FUNCTION_BLOCK AX_TON (* standard timer function block (on-delay timing) *)
  (* Standard: 61499-2; Classification: standard timer function block; Description: Copyright (c) 2024 HR Agrartechnik GmbH This program and the accompanying materials are made available under the terms of the Eclipse Public License 2.0 which is available at https://www.eclipse.org/legal/epl-2.0/ SPDX-License-Identifier: EPL-2.0 *)
  (* Version 3.0, 2025-04-14, Patrick Aigner, changed package *)
  (* Version 1.0, 2024-03-04, Franz Hoepfinger, HR Agrartechnik GmbH *)
  PACKAGE adapter::events::unidirectional::timers;
  IMPORT eclipse4diac::core::TypeHash;
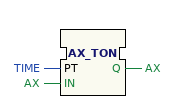
  VAR_INPUT
    PT : TIME; (* Process time *)
  END_VAR
  SOCKETS
    IN : adapter::types::unidirectional::AX; (* Input *)
  END_SOCKETS
  PLUGS
    Q : adapter::types::unidirectional::AX; (* Output *)
  END_PLUGS
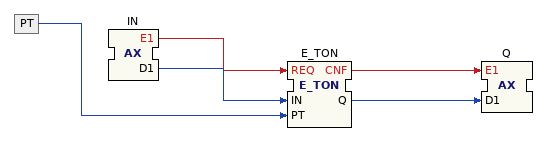
  FBS
    E_TON : iec61499::events::timers::E_TON;
  END_FBS
  EVENT_CONNECTIONS
    E_TON.CNF TO Q.E1;
    IN.E1 TO E_TON.REQ;
  END_CONNECTIONS
  DATA_CONNECTIONS
    E_TON.Q TO Q.D1;
    IN.D1 TO E_TON.IN;
    PT TO E_TON.PT;
  END_CONNECTIONS
END_FUNCTION_BLOCK
